FUNCTION_BLOCK OPCUA_VARIABLE_WRITER
  {SET_ATTRIBUTE(OpcUa, POINT.ENDPOINT)}
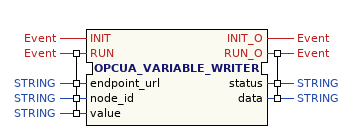
  EVENT_INPUT
    INIT;
    RUN WITH endpoint_url, node_id, value; {SET_ATTRIBUTE(OpcUa, Method)}
  END_EVENT
  EVENT_OUTPUT
    INIT_O;
    RUN_O WITH status, data;
  END_EVENT
  VAR_INPUT
    endpoint_url : STRING; {SET_ATTRIBUTE(OpcUa, Constant)}
    node_id : STRING; {SET_ATTRIBUTE(OpcUa, Constant)}
    value : STRING; {SET_ATTRIBUTE(OpcUa, Constant)}
  END_VAR
  VAR_OUTPUT
    status : STRING; {SET_ATTRIBUTE(OpcUa, Variable)}
    data : STRING; {SET_ATTRIBUTE(OpcUa, Variable)}
  END_VAR
END_FUNCTION_BLOCK
